Staubli VAL3: start.pgx

program start()
begin
  //1.注释不能写在begin上面
  //2.注释不能写在end下面
  //3.语句后面没有分号也没有冒号

  popUpMsg("Hello world")


end
